// TIA Portal V17 export
// export: Created 2025-06-25T13:13:30.5812184Z, ExportSetting WithDefaults, DisplayName Totally Integrated Automation Portal, DisplayVersion V17 Update 8, DisplayName TIA Portal Openness, DisplayVersion V17 Update 8, DisplayName TIA Portal Version Control Interface, DisplayVersion V17, DisplayName STEP 7 Professional, DisplayVersion V17 Update 8, DisplayName STEP 7 Safety, DisplayVersion V17 Update 6, DisplayName WinCC Advanced, DisplayVersion V17 Update 8
TYPE "stProgressivePeriodicRegulator4"
// stored: IsFailsafeCompliant false
   STRUCT
      bEnable : Bool;   // 1 = controller enabled, 0 = disabled
      bFault : Bool;   // 1 = controller fault, 0 = ok
      bOutput : Bool;   // 1 = output active
      bManualOverride : Bool;   // 1 = activate override
      bOverrideCmd : Bool;   // 1 = force output on
      bManualMode : Bool;   // 1 = activate manual mode
      nMode : USInt;   // 0 = Off, 1 = Auto, 2 = Manual, 3 = Manual Override
      tManualPeriod : Time;   // Fixed period
      tOnTime : Time;   // On time of period (duty cycle)
      tPeriod : Time;   // Total period (frequency)
      tOnTimeElapsed : Time;
      tPeriodElapsed : Time;
      fPV : Real;   // Process value
      fPumpSpeed : Real;   // [rpm] Fixed pump speed (hack)
      Param : Struct
         Limit : Array[0..3] of Real;   // Process value thresholds
         Period : Array[0..3] of Time;   // Periods between activations
      END_STRUCT;
   END_STRUCT;
END_TYPE
